FUNCTION F_SubStringSelectedFile : STRING
VAR_INPUT
	sSelectedFile : STRING;
END_VAR
VAR
	
END_VAR

F_SubStringSelectedFile := DELETE(sSelectedFile,2,LEN(sSelectedFile)-1);
F_SubStringSelectedFile := DELETE(F_SubStringSelectedFile,2,0);

END_FUNCTION

(* stored: Version 1.1.0.1, ProductVersion 3.1.4024.6
   POU F_SubStringSelectedFile: Id {202eb4b0-cea0-40bd-a529-01cc062f6f1f}, SpecialFunc None *)
